# EPICS substitutions: ipimbIocApp/Db/ioc-tst-05.substitutions
#==============================================================================
#
# Abs:  IOC Administration Records
#
# Name: iocAdmin.substitutions
#
#==============================================================================
#
file ipimb.template
{
	pattern
	{ RECNAME    , BOX      }
	{ TST:R01:PIM:01 , TST-R01-PIM-01 }
}
